(* Logix 5000 project; controller Test_Bench vendor 1 type 14 code 155 rev 34.11; software revision 34.00 *)

TASK MainTask (continuous, watchdog 500 ms) : MainProgram

MODULES
   Local : vendor 1 type 14 code 155 (PointIO 0, rev 34.11)
      encoder : 842E-CM-M (Ethernet 192.168.100.50, rev 1.1, MotionDiagnostics RPI 1 ms, MotionSync RPI 1 ms)
      servo : vendor 1 type 37 code 49 (Ethernet 192.168.100.194, rev 7.1, MotionSync RPI 1 ms, MotionDiagnostics RPI 1 ms)
      Discrete_IO : Embedded (PointIO 1, rev 34.11, Output RPI 20 ms)
END_MODULES

ADD_ON_INSTRUCTION AL2xxx_8PORT_ConfigOnly   (* revision 1.0, vendor ifm efector *)
// Revision note:
// Use with any IO-link hub for config of Equip ID, Device Status and factory reset functions.
VAR_IN_OUT
   PLC_Input : INT[223]; {required}
   PLC_Output : INT[151]; {required}
        [5].7   // Trigger Bit for all commands
END_VAR
VAR_OUTPUT
   IOL_Mode : BOOL; {access Read Only, visible}
   Device_Not_Connected : BOOL; {access Read Only, visible}
END_VAR
VAR_IN_OUT
   IOLinkMaster_Name : DINT; {required}   // Used to control AL1x2x_Cmd_Ry output bit. Is use by any AOI with commands on the same IO-Link Master
END_VAR
VAR_OUTPUT
   TimeOut : BOOL;
   Invalid_Data : BOOL; {access Read Only, visible}
   Wrong_VID_DID : BOOL; {access Read Only, visible}   // Indication when Automatic Device Repl detects a differenet Vendor ID or Device ID
   AOI_Settings_Error : BOOL; {visible}
   AL1x2x_Cmd_Rdy : BOOL; {visible}   // If HI comman can be sent to device. If Low no command can be sent
   Config_Cmds_Busy : BOOL; {visible}   // Commands are processing
   Config_Cmds_DN : BOOL; {visible}
END_VAR
VAR_INPUT
   Port_Number : INT; {visible}
END_VAR
VAR_OUTPUT
   Vendor_ID : INT; {access Read Only, visible}
   Device_ID : DINT; {access Read Only, visible}
END_VAR
VAR_INPUT
   Set_Equipment_Spec_ID : INT; {visible}   // Value Range 0-127
   ConfigCmd_Trigger : BOOL; {visible}   // Command to send configuaration parameters
END_VAR
VAR_IN_OUT
   Config_CmdsResp_Buffer : INT[3]; {required}
        [0]   // Resp Write Equipment Specfic ID
        [1]   // Resp Read Equipment Specific ID
END_VAR
VAR_INPUT
   DeviceStatus_Trigger : BOOL; {visible}   // Command to get Short Circuits by port number
END_VAR
VAR_OUTPUT
   DeviceStatus_DN : BOOL; {access Read Only, visible}
END_VAR
VAR_INPUT
   Factory_Reset_Trigger : BOOL; {visible}
END_VAR
VAR_OUTPUT
   Factory_Reset_DN : BOOL; {access None, visible}
   Device_Ok : BOOL; {access Read Only, visible}   // Latched after Device Status Trigger and Cmds_DN
   Maintenance_required : BOOL; {access Read Only}
   Out_of_specifications : BOOL; {access Read Only, visible}   // Supply power under-run
   Functional_check : BOOL; {access Read Only, visible}   // Short Circuit
   Failure : BOOL; {access Read Only}
END_VAR
VAR
   Offset_StatusFlgs : INT; {access None}
   RealPort_Num : INT; {access None}
   StatusFlgs_Offset : INT; {access None}
   PLCTrigger : SINT; {access None}   // Local SINT to set the trigger of an acyclic command (PLCInput[5].7
   Device_Status : SINT; {access Read Only}
   AOI_Port_Error : BOOL; {access None}   // When set no commands are allowed
   AOI_Trigger_Error : BOOL; {access None}   // Signal to Latch when both Config and Recipe Change triggers are set high
   DevNotConn_Signal : BOOL; {access None}   // Latch signal set by Device Not Connected bit
   AL1x2x_Cmd_Rdy_Timer : TIMER := (PRE := 20); {access None}
   Factory_Reset_Lch : BOOL; {access None}   // Latched by trigger to hold trigger high until commands are done.
   ConfigCmd_Lch : BOOL; {access None}   // Latched by trigger to hold trigger high until commands are done.
   TriggerCmdBuffer_ONS : BOOL; {access None}
   Factory_ResetDN_Signal : BOOL; {access None}
   Skip_Cmd0 : BOOL; {access None}
   Cmd2TriggerDelay : TIMER := (PRE := 20); {access None}
   Cmd2ReleaseTrigger : BOOL; {access None}
   Cmd2_Trigger : BOOL; {access None}
   Cmd2_DN_Error : BOOL; {access None}
   Cmd2_DN : BOOL; {access None}
   Cmd2_Busy : BOOL; {access None}
   Cmd2 : BOOL; {access None}
   Cmd1TriggerDelay : TIMER := (PRE := 20); {access None}
   Cmd1ReleaseTrigger : BOOL; {access None}
   Cmd1_Trigger : BOOL; {access None}
   Cmd1_PLC_OutTrigger : BOOL; {access None}
   Cmd1_DN_Error : BOOL; {access None}
   Cmd1_DN : BOOL; {access None}
   Cmd1_Busy : BOOL; {access None}
   Cmd1 : BOOL; {access None}
   Cmd0ReleaseTrigger : BOOL; {access None}
   Cmd0_Trigger : BOOL; {access None}
   Cmd0_PLC_OutTrigger : BOOL; {access None}
   Cmd0_DN_Error : BOOL; {access None}
   Cmd0_DN : BOOL; {access None}
   Cmd0_Busy : BOOL; {access None}
   Cmd0 : BOOL; {access None}
   Cmd_Array_Empty : INT[16]; {access None}
   TimeOut3 : TIMER := (PRE := 6000); {access None}
   TimeOut2 : TIMER := (PRE := 6000); {access None}   // When RPI time is set > 10ms. Timeout so logic does not get stuck
   TimeOut1 : TIMER := (PRE := 6000); {access None}   // If more than one trigger is sent to mailbox. When timer runs and triggers set low the logic will reset.
   TimeOut3_Signal : BOOL; {access None}
   TimeOut2_Signal : BOOL; {access None}
   TimeOut1_Signal : BOOL; {access None}
   DeviceStatus_Lch : BOOL; {access None}   // Latched by trigger to hold trigger high until commands are done.
   DeviceStatus_CmdDN_Signal : BOOL; {access None}
   ResetCmd : BOOL; {access None}   // Read a command so that the PLC_Input[3] is reset to <>2
   NotAppInput_Array10 : INT[10] := ([0] := -32640, [1] := -32640, [2] := -32640, [3] := -32640, [4] := -32640, [5] := -32640, [6] := -32640, [7] := -32640, [8] := -32640, [9] := -32640); {access None}   // Fills the N/A fields -128 value
END_VAR

ROUTINE Logic   (* ladder *)
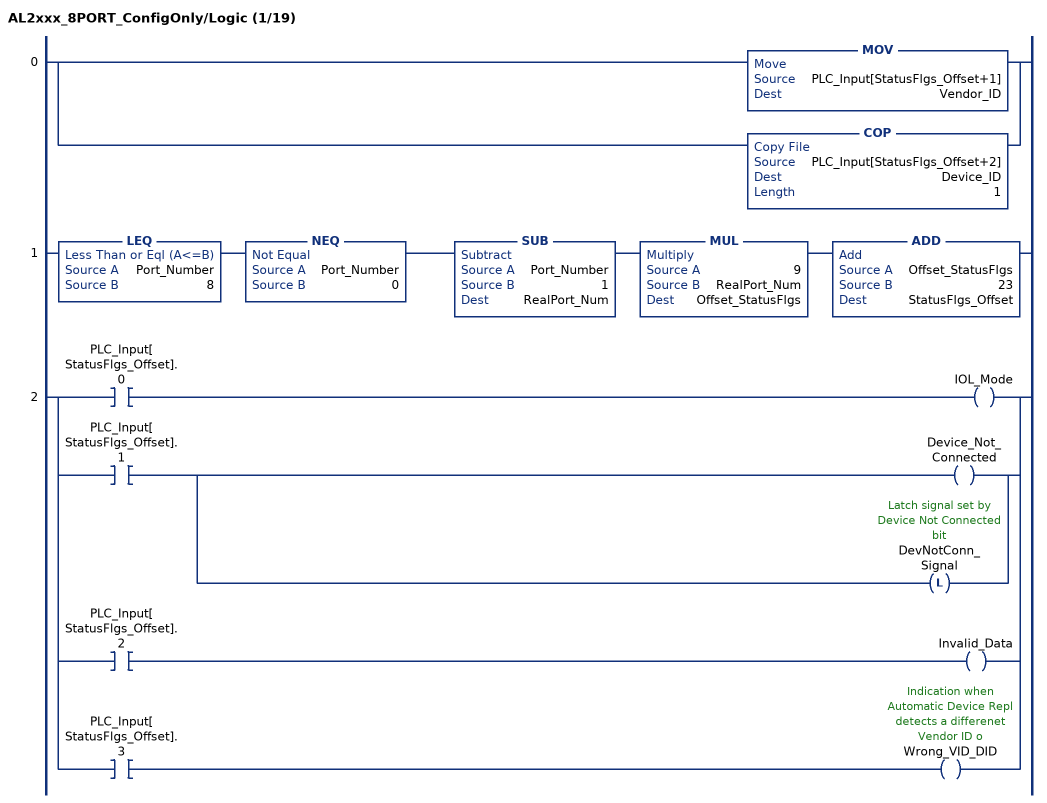
   0: [MOV(PLC_Input[StatusFlgs_Offset+1],Vendor_ID) ,COP(PLC_Input[StatusFlgs_Offset+2],Device_ID,1) ];
   1: LEQ(Port_Number,8)NEQ(Port_Number,0)SUB(Port_Number,1,RealPort_Num)MUL(9,RealPort_Num,Offset_StatusFlgs)ADD(Offset_StatusFlgs,23,StatusFlgs_Offset);
   2: [XIC(PLC_Input[StatusFlgs_Offset].0) OTE(IOL_Mode) ,XIC(PLC_Input[StatusFlgs_Offset].1) [OTE(Device_Not_Connected) ,OTL(DevNotConn_Signal) ] ,XIC(PLC_Input[StatusFlgs_Offset].2) OTE(Invalid_Data) ,XIC(PLC_Input[StatusFlgs_Offset].3) OTE(Wrong_VID_DID) ];
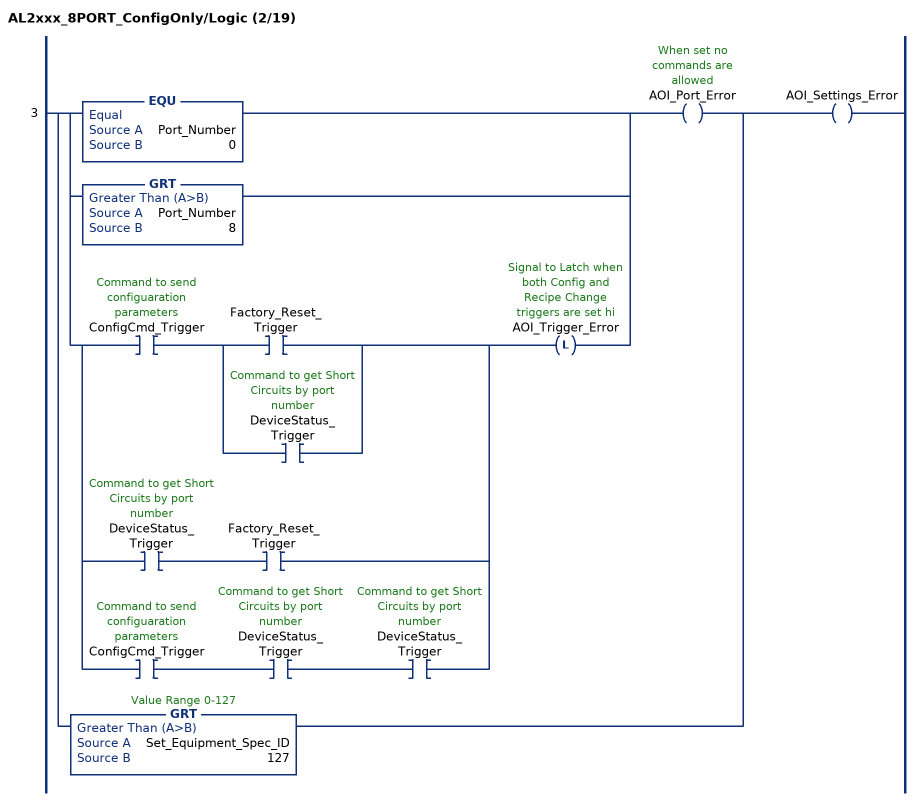
   3: [[EQU(Port_Number,0) ,GRT(Port_Number,8) ,[XIC(ConfigCmd_Trigger) [XIC(Factory_Reset_Trigger) ,XIC(DeviceStatus_Trigger) ] ,XIC(DeviceStatus_Trigger) XIC(Factory_Reset_Trigger) ,XIC(ConfigCmd_Trigger) XIC(DeviceStatus_Trigger) XIC(DeviceStatus_Trigger) ] OTL(AOI_Trigger_Error) ] OTE(AOI_Port_Error) ,GRT(Set_Equipment_Spec_ID,127) ]OTE(AOI_Settings_Error);
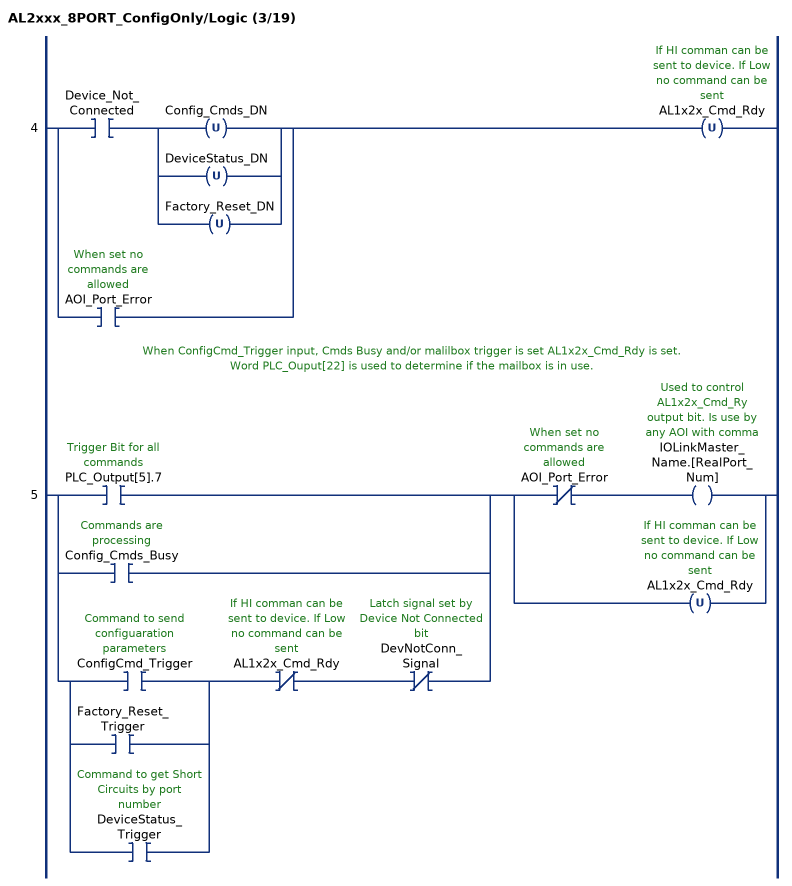
   4: [XIC(Device_Not_Connected) [OTU(Config_Cmds_DN) ,OTU(DeviceStatus_DN) ,OTU(Factory_Reset_DN) ] ,XIC(AOI_Port_Error) ]OTU(AL1x2x_Cmd_Rdy);
   // When ConfigCmd_Trigger input, Cmds Busy and/or malilbox trigger is set AL1x2x_Cmd_Rdy is set.
   // Word PLC_Ouput[22] is used to determine if the mailbox is in use.
   5: [XIC(PLC_Output[5].7) ,XIC(Config_Cmds_Busy) ,[XIC(ConfigCmd_Trigger) ,XIC(Factory_Reset_Trigger) ,XIC(DeviceStatus_Trigger) ] XIO(AL1x2x_Cmd_Rdy) XIO(DevNotConn_Signal) ][XIO(AOI_Port_Error) OTE(IOLinkMaster_Name.[RealPort_Num]) ,OTU(AL1x2x_Cmd_Rdy) ];
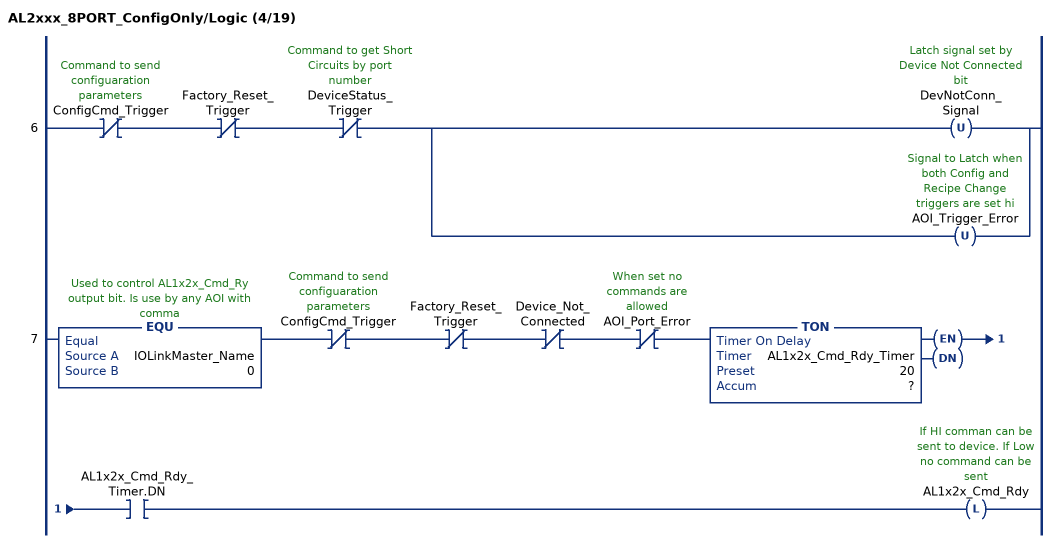
   6: XIO(ConfigCmd_Trigger)XIO(Factory_Reset_Trigger)XIO(DeviceStatus_Trigger)[OTU(DevNotConn_Signal) ,OTU(AOI_Trigger_Error) ];
   7: EQU(IOLinkMaster_Name,0)XIO(ConfigCmd_Trigger)XIO(Factory_Reset_Trigger)XIO(Device_Not_Connected)XIO(AOI_Port_Error)TON(AL1x2x_Cmd_Rdy_Timer,?,?)XIC(AL1x2x_Cmd_Rdy_Timer.DN)OTL(AL1x2x_Cmd_Rdy);
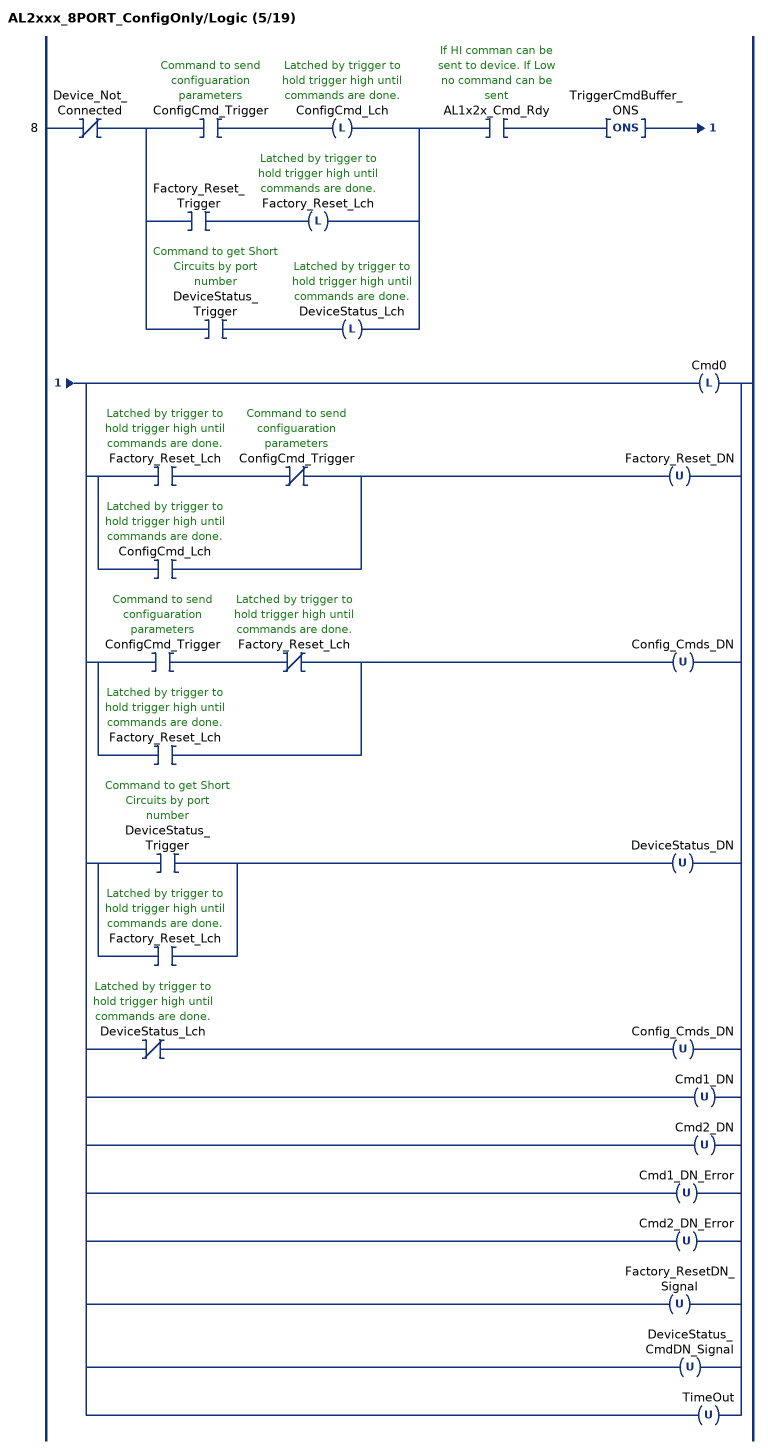
   8: XIO(Device_Not_Connected)[XIC(ConfigCmd_Trigger) OTL(ConfigCmd_Lch) ,XIC(Factory_Reset_Trigger) OTL(Factory_Reset_Lch) ,XIC(DeviceStatus_Trigger) OTL(DeviceStatus_Lch) ]XIC(AL1x2x_Cmd_Rdy)ONS(TriggerCmdBuffer_ONS)[OTL(Cmd0) ,[XIC(Factory_Reset_Lch) XIO(ConfigCmd_Trigger) ,XIC(ConfigCmd_Lch) ] OTU(Factory_Reset_DN) ,[XIC(ConfigCmd_Trigger) XIO(Factory_Reset_Lch) ,XIC(Factory_Reset_Lch) ] OTU(Config_Cmds_DN) ,[XIC(DeviceStatus_Trigger) ,XIC(Factory_Reset_Lch) ] OTU(DeviceStatus_DN) ,XIO(DeviceStatus_Lch) OTU(Config_Cmds_DN) ,OTU(Cmd1_DN) ,OTU(Cmd2_DN) ,OTU(Cmd1_DN_Error) ,OTU(Cmd2_DN_Error) ,OTU(Factory_ResetDN_Signal) ,OTU(DeviceStatus_CmdDN_Signal) ,OTU(TimeOut) ];
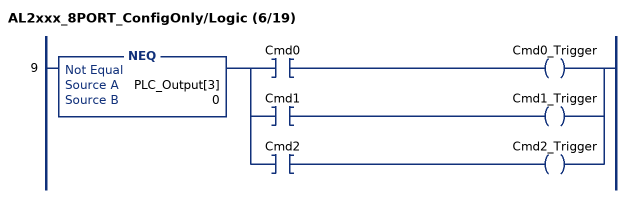
   9: NEQ(PLC_Output[3],0)[XIC(Cmd0) OTE(Cmd0_Trigger) ,XIC(Cmd1) OTE(Cmd1_Trigger) ,XIC(Cmd2) OTE(Cmd2_Trigger) ];
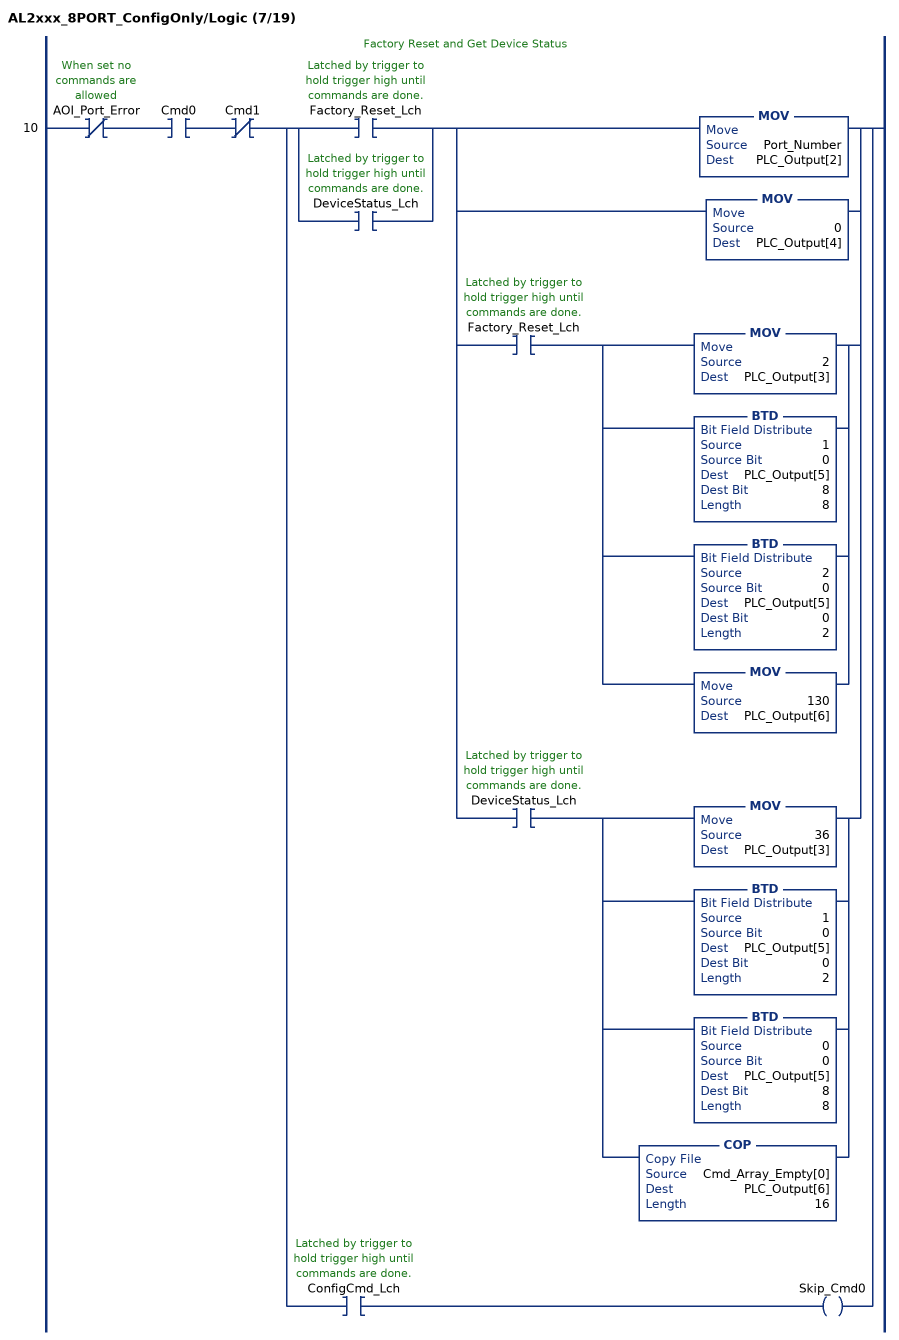
   // Factory Reset and Get Device Status
   10: XIO(AOI_Port_Error)XIC(Cmd0)XIO(Cmd1)[[XIC(Factory_Reset_Lch) ,XIC(DeviceStatus_Lch) ] [MOV(Port_Number,PLC_Output[2]) ,MOV(0,PLC_Output[4]) ,[XIC(Factory_Reset_Lch) [MOV(2,PLC_Output[3]) ,BTD(1,0,PLC_Output[5],8,8) ,BTD(2,0,PLC_Output[5],0,2) ,MOV(130,PLC_Output[6]) ] ,XIC(DeviceStatus_Lch) [MOV(36,PLC_Output[3]) ,BTD(1,0,PLC_Output[5],0,2) ,BTD(0,0,PLC_Output[5],8,8) ,COP(Cmd_Array_Empty[0],PLC_Output[6],16) ] ] ] ,XIC(ConfigCmd_Lch) OTE(Skip_Cmd0) ];
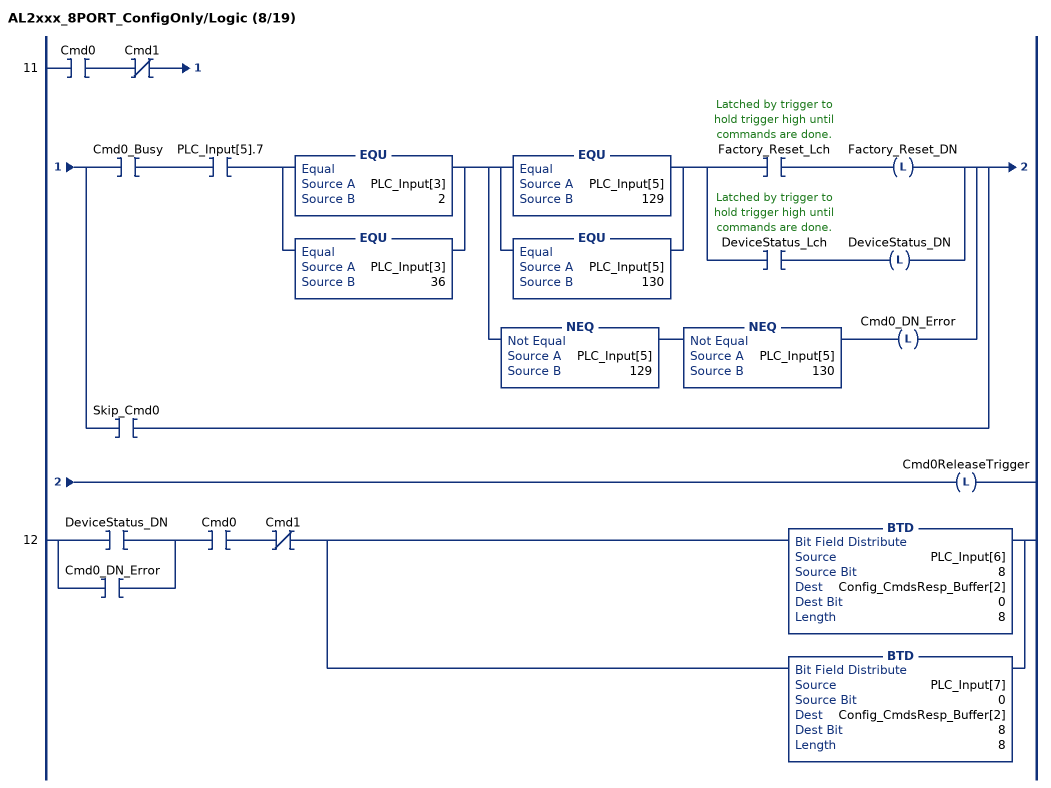
   11: XIC(Cmd0)XIO(Cmd1)[XIC(Cmd0_Busy) XIC(PLC_Input[5].7) [EQU(PLC_Input[3],2) ,EQU(PLC_Input[3],36) ] [[EQU(PLC_Input[5],129) ,EQU(PLC_Input[5],130) ] [XIC(Factory_Reset_Lch) OTL(Factory_Reset_DN) ,XIC(DeviceStatus_Lch) OTL(DeviceStatus_DN) ] ,NEQ(PLC_Input[5],129) NEQ(PLC_Input[5],130) OTL(Cmd0_DN_Error) ] ,XIC(Skip_Cmd0) ]OTL(Cmd0ReleaseTrigger);
   12: [XIC(DeviceStatus_DN) ,XIC(Cmd0_DN_Error) ]XIC(Cmd0)XIO(Cmd1)[BTD(PLC_Input[6],8,Config_CmdsResp_Buffer[2],0,8) ,BTD(PLC_Input[7],0,Config_CmdsResp_Buffer[2],8,8) ];
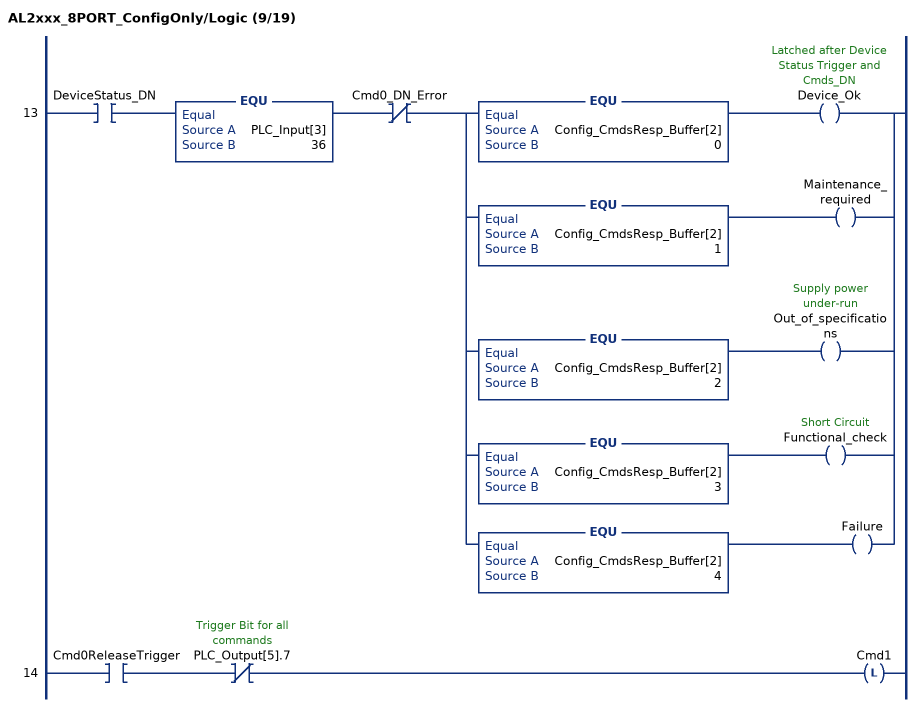
   13: XIC(DeviceStatus_DN)EQU(PLC_Input[3],36)XIO(Cmd0_DN_Error)[EQU(Config_CmdsResp_Buffer[2],0) OTE(Device_Ok) ,EQU(Config_CmdsResp_Buffer[2],1) OTE(Maintenance_required) ,EQU(Config_CmdsResp_Buffer[2],2) OTE(Out_of_specifications) ,EQU(Config_CmdsResp_Buffer[2],3) OTE(Functional_check) ,EQU(Config_CmdsResp_Buffer[2],4) OTE(Failure) ];
   14: XIC(Cmd0ReleaseTrigger)XIO(PLC_Output[5].7)OTL(Cmd1);
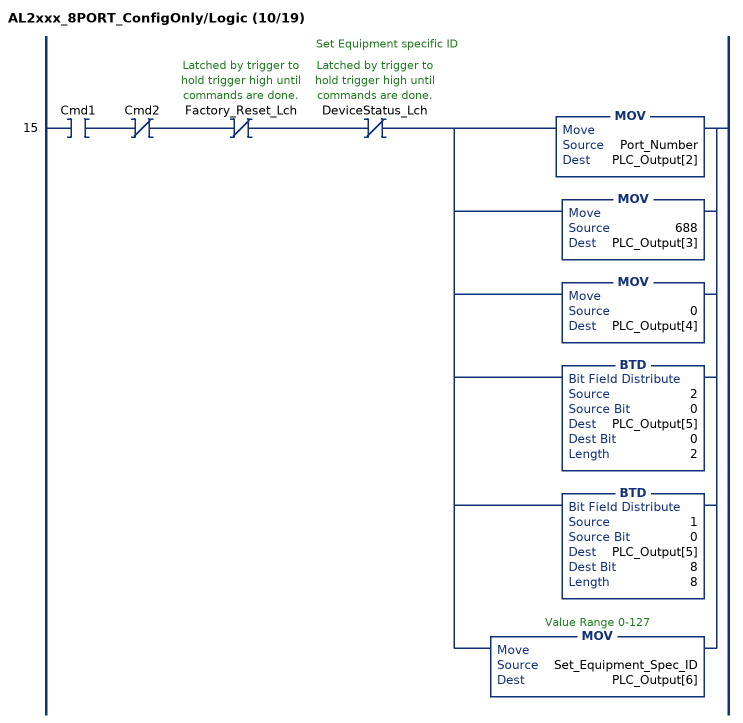
   // Set Equipment specific ID
   15: XIC(Cmd1)XIO(Cmd2)XIO(Factory_Reset_Lch)XIO(DeviceStatus_Lch)[MOV(Port_Number,PLC_Output[2]) ,MOV(688,PLC_Output[3]) ,MOV(0,PLC_Output[4]) ,BTD(2,0,PLC_Output[5],0,2) ,BTD(1,0,PLC_Output[5],8,8) ,MOV(Set_Equipment_Spec_ID,PLC_Output[6]) ];
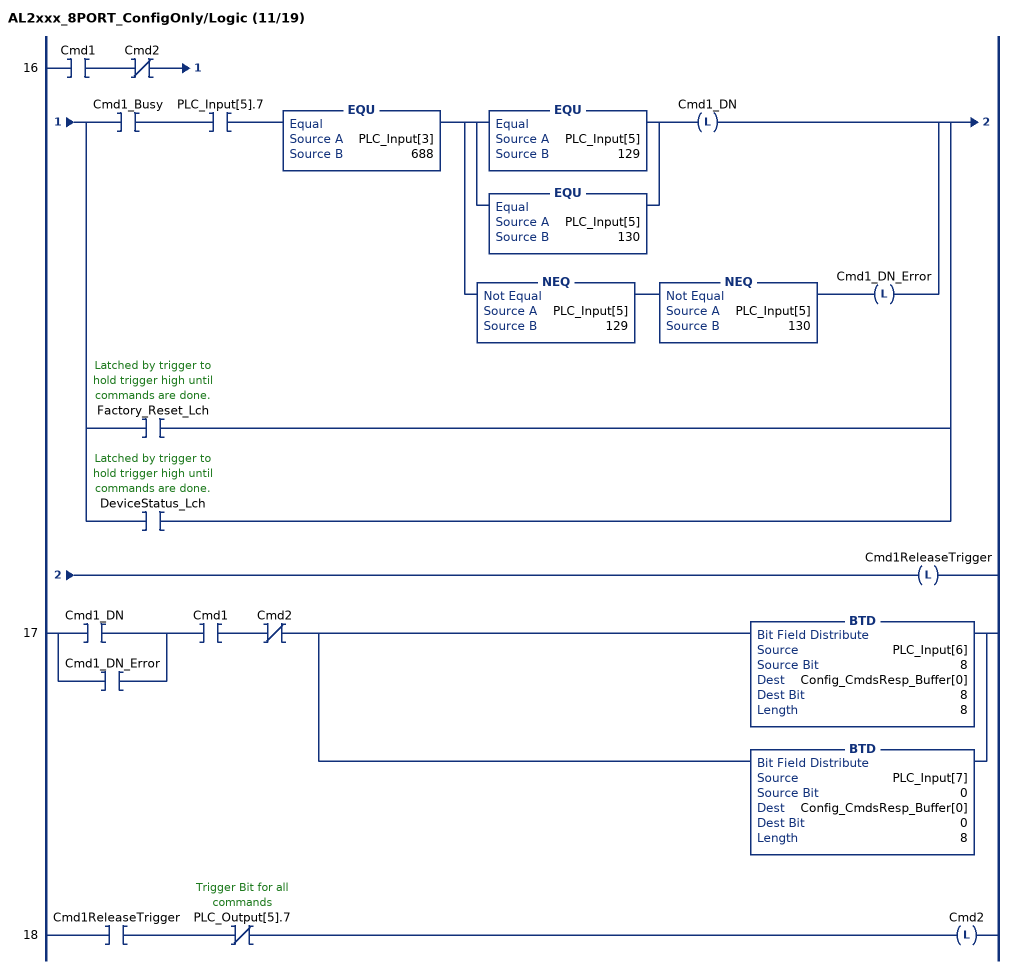
   16: XIC(Cmd1)XIO(Cmd2)[XIC(Cmd1_Busy) XIC(PLC_Input[5].7) EQU(PLC_Input[3],688) [[EQU(PLC_Input[5],129) ,EQU(PLC_Input[5],130) ] OTL(Cmd1_DN) ,NEQ(PLC_Input[5],129) NEQ(PLC_Input[5],130) OTL(Cmd1_DN_Error) ] ,[XIC(Factory_Reset_Lch) ,XIC(DeviceStatus_Lch) ] ]OTL(Cmd1ReleaseTrigger);
   17: [XIC(Cmd1_DN) ,XIC(Cmd1_DN_Error) ]XIC(Cmd1)XIO(Cmd2)[BTD(PLC_Input[6],8,Config_CmdsResp_Buffer[0],8,8) ,BTD(PLC_Input[7],0,Config_CmdsResp_Buffer[0],0,8) ];
   18: XIC(Cmd1ReleaseTrigger)XIO(PLC_Output[5].7)OTL(Cmd2);
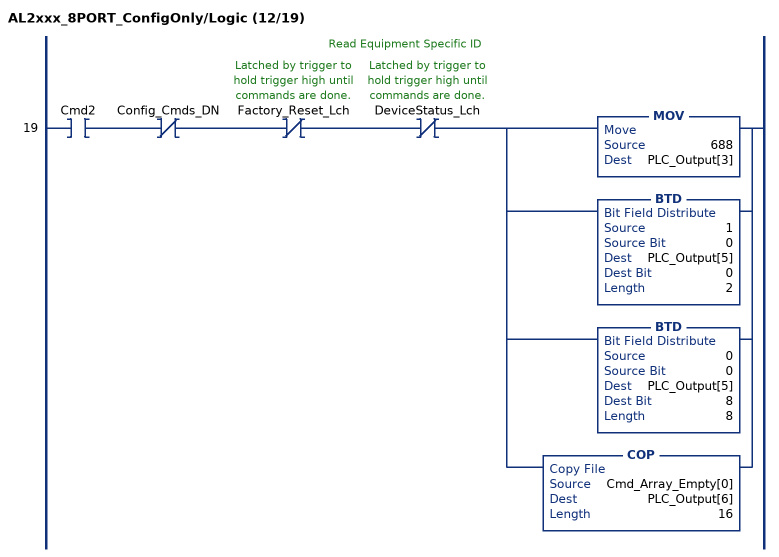
   // Read Equipment Specific ID
   19: XIC(Cmd2)XIO(Config_Cmds_DN)XIO(Factory_Reset_Lch)XIO(DeviceStatus_Lch)[MOV(688,PLC_Output[3]) ,BTD(1,0,PLC_Output[5],0,2) ,BTD(0,0,PLC_Output[5],8,8) ,COP(Cmd_Array_Empty[0],PLC_Output[6],16) ];
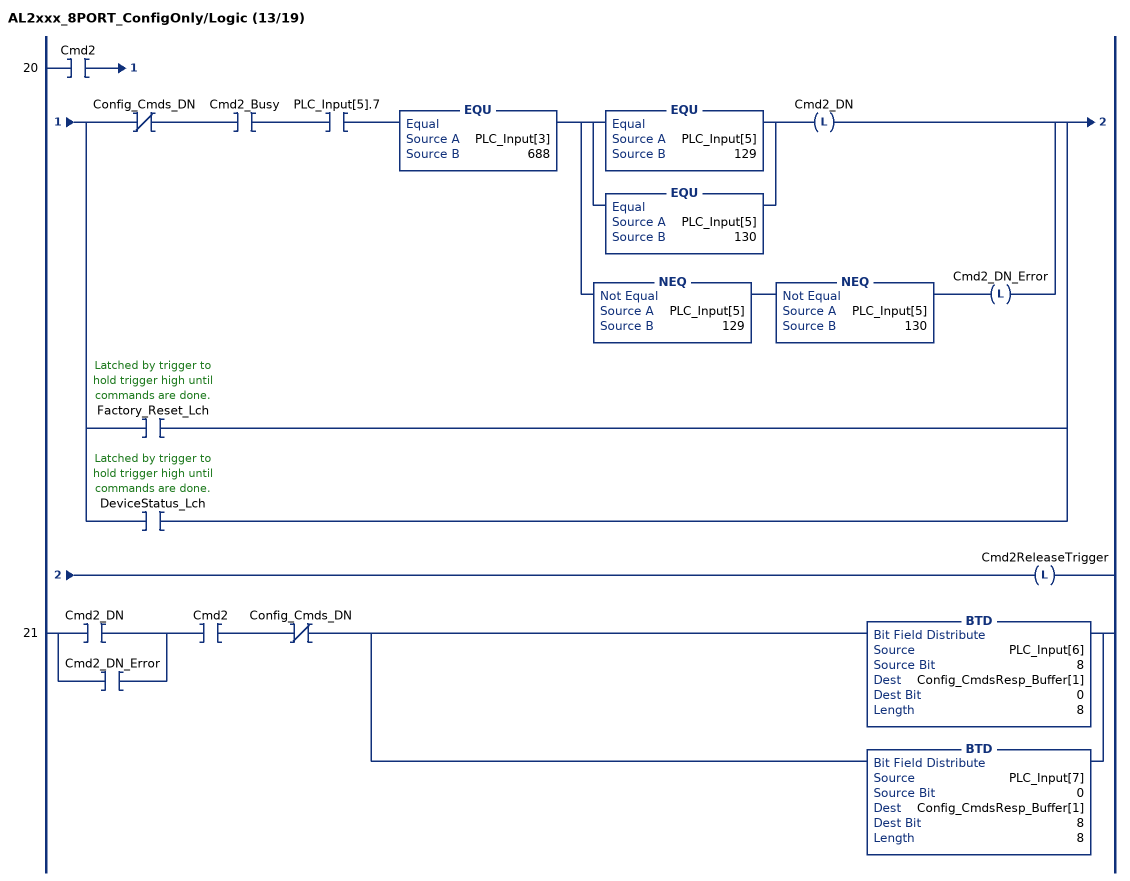
   20: XIC(Cmd2)[XIO(Config_Cmds_DN) XIC(Cmd2_Busy) XIC(PLC_Input[5].7) EQU(PLC_Input[3],688) [[EQU(PLC_Input[5],129) ,EQU(PLC_Input[5],130) ] OTL(Cmd2_DN) ,NEQ(PLC_Input[5],129) NEQ(PLC_Input[5],130) OTL(Cmd2_DN_Error) ] ,[XIC(Factory_Reset_Lch) ,XIC(DeviceStatus_Lch) ] ]OTL(Cmd2ReleaseTrigger);
   21: [XIC(Cmd2_DN) ,XIC(Cmd2_DN_Error) ]XIC(Cmd2)XIO(Config_Cmds_DN)[BTD(PLC_Input[6],8,Config_CmdsResp_Buffer[1],0,8) ,BTD(PLC_Input[7],0,Config_CmdsResp_Buffer[1],8,8) ];
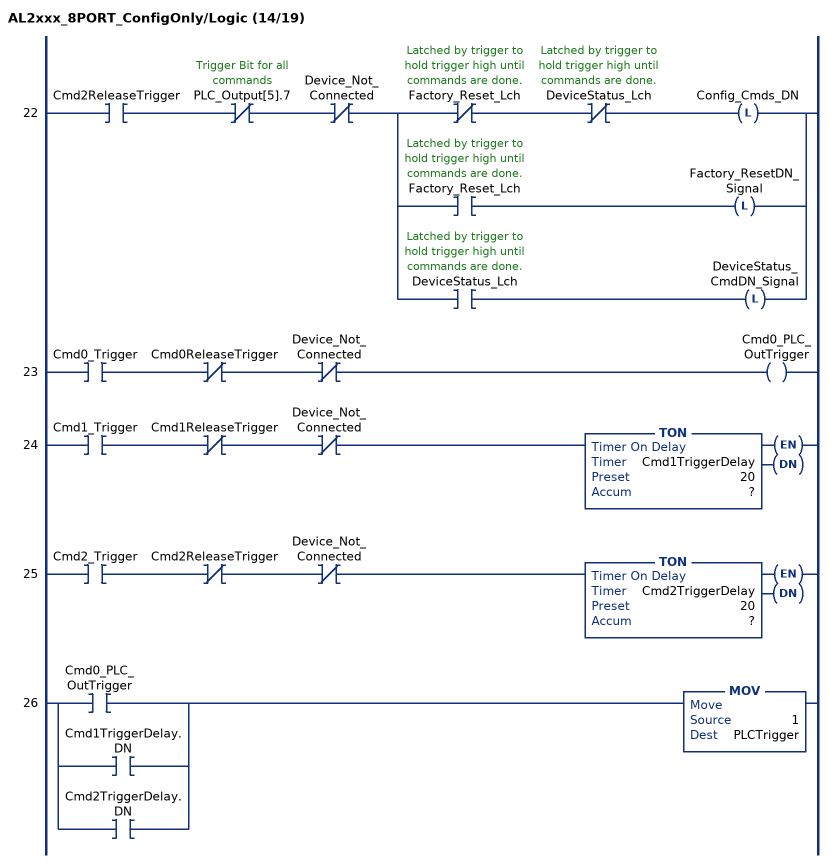
   22: XIC(Cmd2ReleaseTrigger)XIO(PLC_Output[5].7)XIO(Device_Not_Connected)[XIO(Factory_Reset_Lch) XIO(DeviceStatus_Lch) OTL(Config_Cmds_DN) ,XIC(Factory_Reset_Lch) OTL(Factory_ResetDN_Signal) ,XIC(DeviceStatus_Lch) OTL(DeviceStatus_CmdDN_Signal) ];
   23: XIC(Cmd0_Trigger)XIO(Cmd0ReleaseTrigger)XIO(Device_Not_Connected)OTE(Cmd0_PLC_OutTrigger);
   24: XIC(Cmd1_Trigger)XIO(Cmd1ReleaseTrigger)XIO(Device_Not_Connected)TON(Cmd1TriggerDelay,?,?);
   25: XIC(Cmd2_Trigger)XIO(Cmd2ReleaseTrigger)XIO(Device_Not_Connected)TON(Cmd2TriggerDelay,?,?);
   26: [XIC(Cmd0_PLC_OutTrigger) ,XIC(Cmd1TriggerDelay.DN) ,XIC(Cmd2TriggerDelay.DN) ]MOV(1,PLCTrigger);
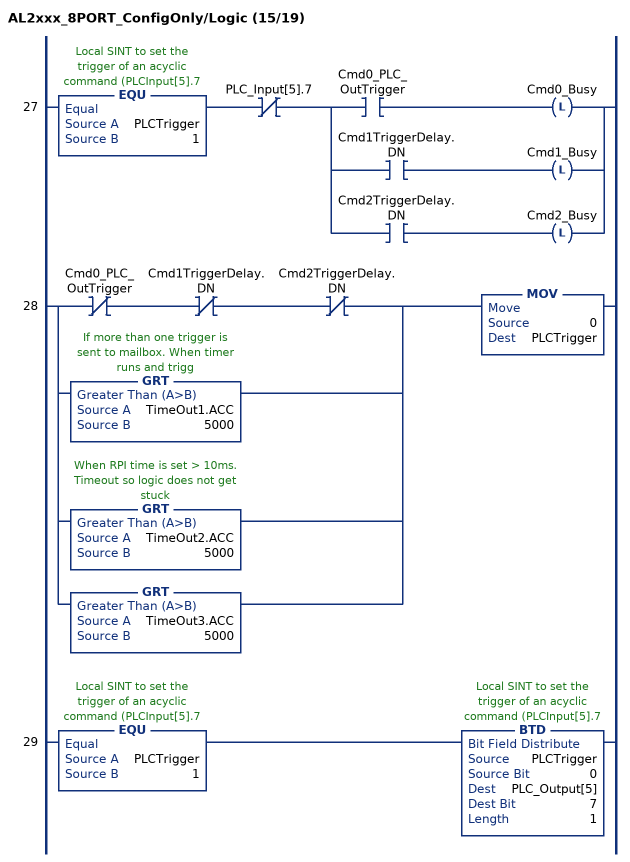
   27: EQU(PLCTrigger,1)XIO(PLC_Input[5].7)[XIC(Cmd0_PLC_OutTrigger) OTL(Cmd0_Busy) ,XIC(Cmd1TriggerDelay.DN) OTL(Cmd1_Busy) ,XIC(Cmd2TriggerDelay.DN) OTL(Cmd2_Busy) ];
   28: [XIO(Cmd0_PLC_OutTrigger) XIO(Cmd1TriggerDelay.DN) XIO(Cmd2TriggerDelay.DN) ,GRT(TimeOut1.ACC,5000) ,GRT(TimeOut2.ACC,5000) ,GRT(TimeOut3.ACC,5000) ]MOV(0,PLCTrigger);
   29: EQU(PLCTrigger,1)BTD(PLCTrigger,0,PLC_Output[5],7,1);
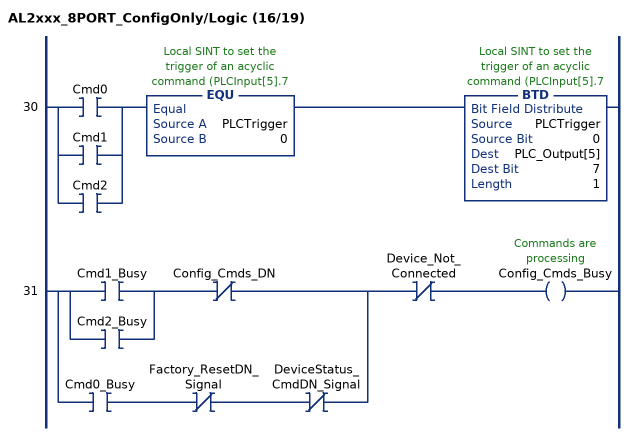
   30: [XIC(Cmd0) ,XIC(Cmd1) ,XIC(Cmd2) ]EQU(PLCTrigger,0)BTD(PLCTrigger,0,PLC_Output[5],7,1);
   31: [[XIC(Cmd1_Busy) ,XIC(Cmd2_Busy) ] XIO(Config_Cmds_DN) ,XIC(Cmd0_Busy) XIO(Factory_ResetDN_Signal) XIO(DeviceStatus_CmdDN_Signal) ]XIO(Device_Not_Connected)OTE(Config_Cmds_Busy);
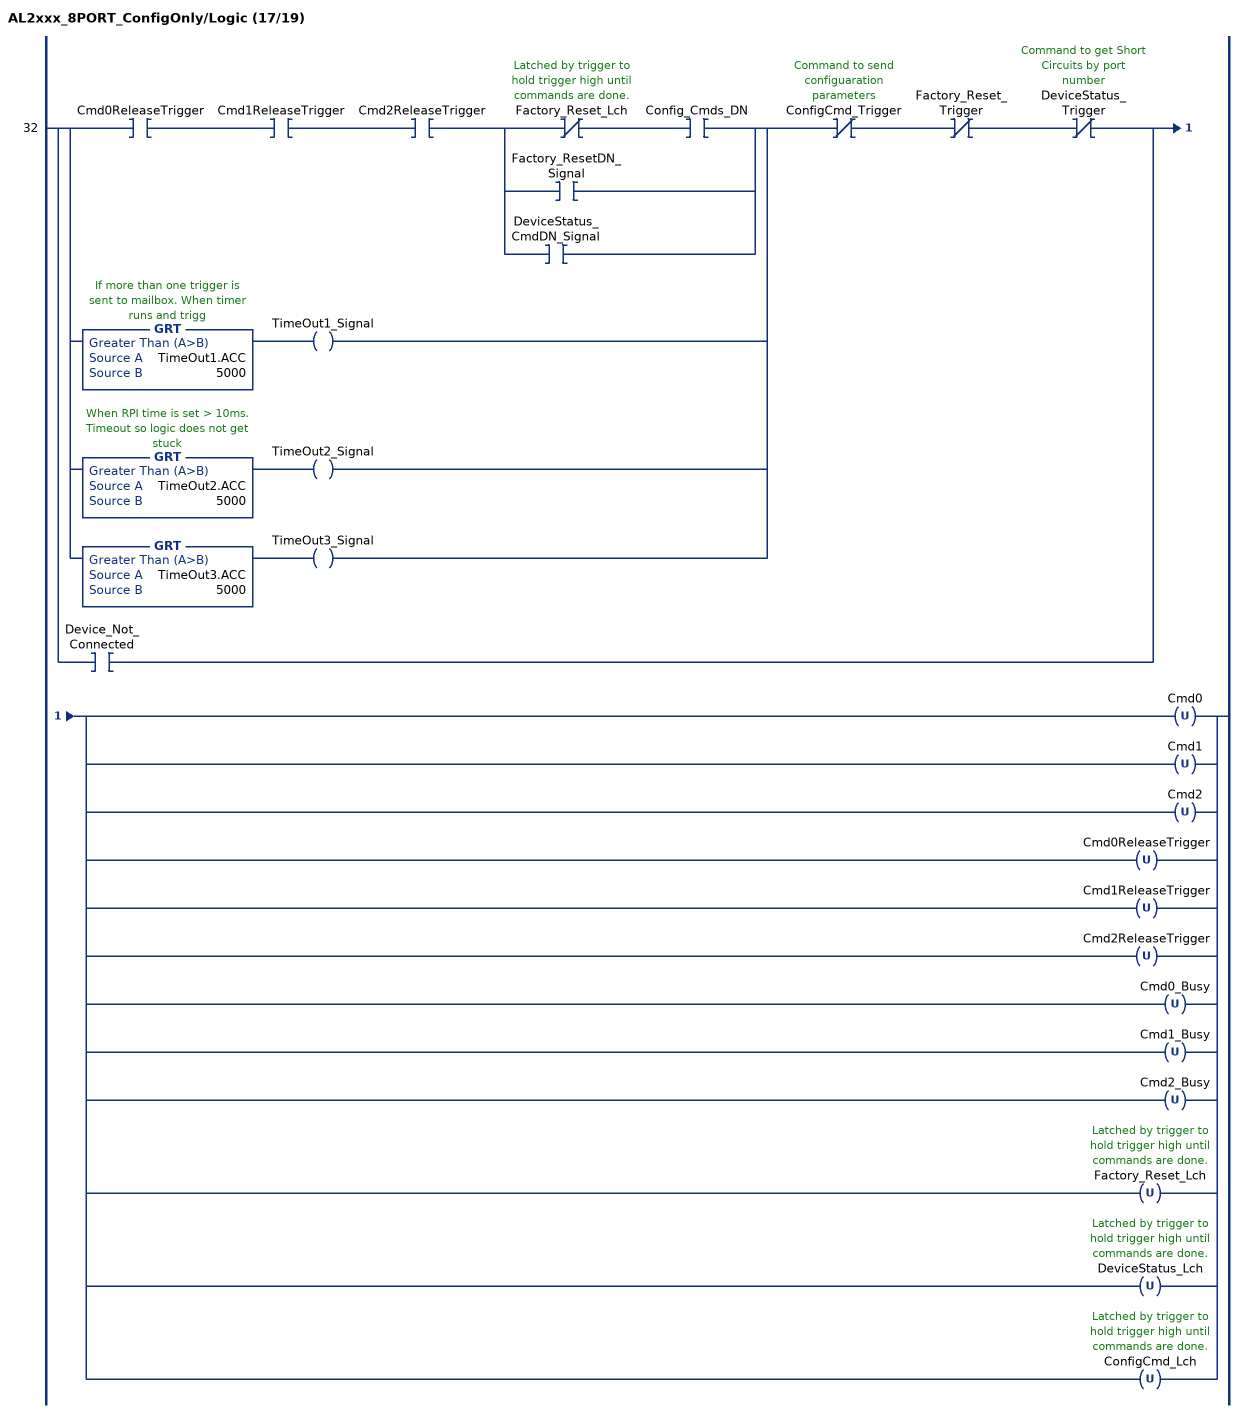
   32: [[XIC(Cmd0ReleaseTrigger) XIC(Cmd1ReleaseTrigger) XIC(Cmd2ReleaseTrigger) [XIO(Factory_Reset_Lch) XIC(Config_Cmds_DN) ,XIC(Factory_ResetDN_Signal) ,XIC(DeviceStatus_CmdDN_Signal) ] ,[GRT(TimeOut1.ACC,5000) OTE(TimeOut1_Signal) ,GRT(TimeOut2.ACC,5000) OTE(TimeOut2_Signal) ,GRT(TimeOut3.ACC,5000) OTE(TimeOut3_Signal) ] ] XIO(ConfigCmd_Trigger) XIO(Factory_Reset_Trigger) XIO(DeviceStatus_Trigger) ,XIC(Device_Not_Connected) ][OTU(Cmd0) ,OTU(Cmd1) ,OTU(Cmd2) ,OTU(Cmd0ReleaseTrigger) ,OTU(Cmd1ReleaseTrigger) ,OTU(Cmd2ReleaseTrigger) ,OTU(Cmd0_Busy) ,OTU(Cmd1_Busy) ,OTU(Cmd2_Busy) ,OTU(Factory_Reset_Lch) ,OTU(DeviceStatus_Lch) ,OTU(ConfigCmd_Lch) ];
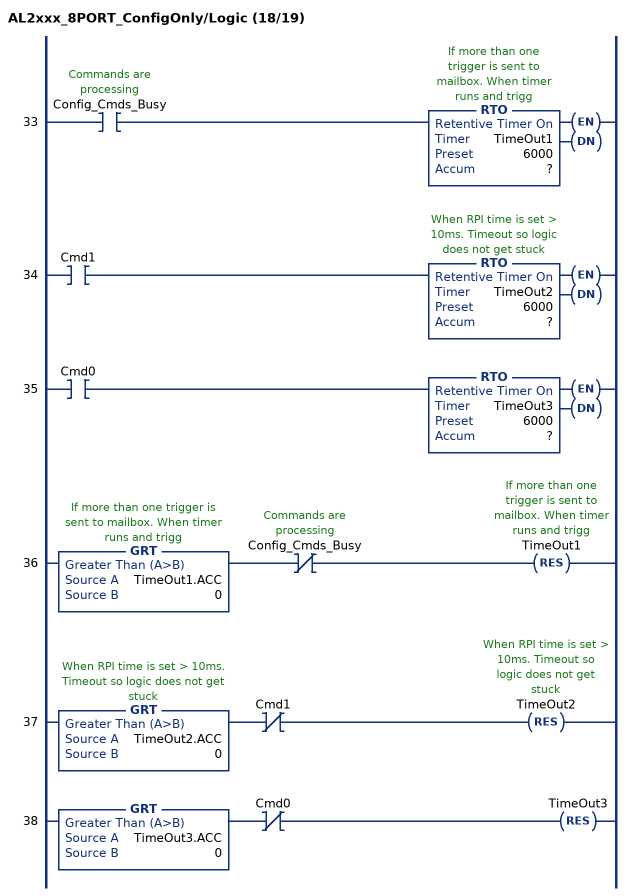
   33: XIC(Config_Cmds_Busy)RTO(TimeOut1,?,?);
   34: XIC(Cmd1)RTO(TimeOut2,?,?);
   35: XIC(Cmd0)RTO(TimeOut3,?,?);
   36: GRT(TimeOut1.ACC,0)XIO(Config_Cmds_Busy)RES(TimeOut1);
   37: GRT(TimeOut2.ACC,0)XIO(Cmd1)RES(TimeOut2);
   38: GRT(TimeOut3.ACC,0)XIO(Cmd0)RES(TimeOut3);
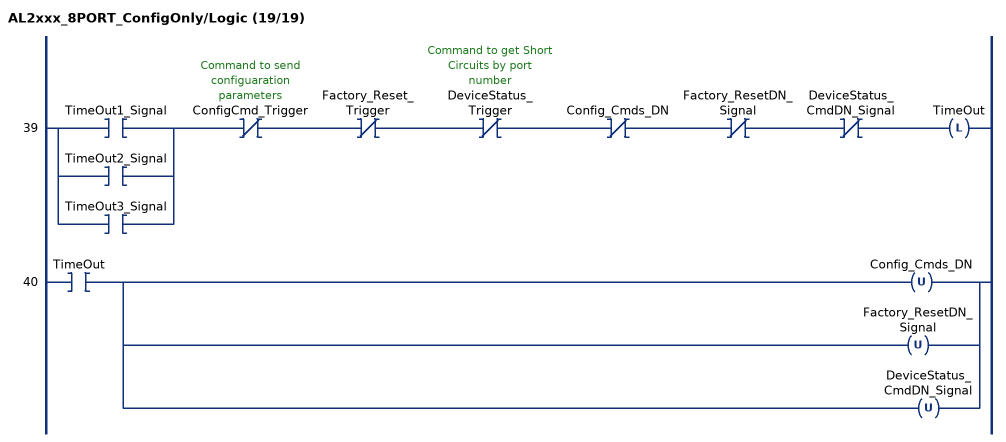
   39: [XIC(TimeOut1_Signal) ,XIC(TimeOut2_Signal) ,XIC(TimeOut3_Signal) ]XIO(ConfigCmd_Trigger)XIO(Factory_Reset_Trigger)XIO(DeviceStatus_Trigger)XIO(Config_Cmds_DN)XIO(Factory_ResetDN_Signal)XIO(DeviceStatus_CmdDN_Signal)OTL(TimeOut);
   40: XIC(TimeOut)[OTU(Config_Cmds_DN) ,OTU(Factory_ResetDN_Signal) ,OTU(DeviceStatus_CmdDN_Signal) ];
END_ROUTINE
END_ADD_ON_INSTRUCTION
